% RSLogix 500 project Sesion13_Tarea1_Josue Santana Robledo Corona.RSS, saved by version 8.40.00.08 %
PROJECT "UNTITLED"    % processor: MicroLogix 1200 %

PROGRAM FILES
  LAD 2 "MAIN"  7 rungs
  LAD 3 "ENTRADAS"  7 rungs
  LAD 4 "SALIDAS"  6 rungs
  LAD 5 "MANUAL"  6 rungs
  LAD 6 "AUTOMATICO"  17 rungs
  LAD 7 "HMI"  1 rungs
  LAD 8 "ALARMAS"  1 rungs
  LAD 9 "LS"  4 rungs
  LAD 10 "PARPADEOS"  5 rungs
  LAD 11 "RESET"  3 rungs

DATA FILES
  O0 OUTPUT  4 elements
  I1 INPUT  4 elements
  S2 STATUS  66 elements
  B3 BINARY  4 elements
  T4 TIMER  8 elements
  C5 COUNTER  3 elements
  R6 CONTROL  1 elements
  N7 INTEGER  1 elements
  F8 FLOAT  1 elements

LADDER 2 "MAIN"
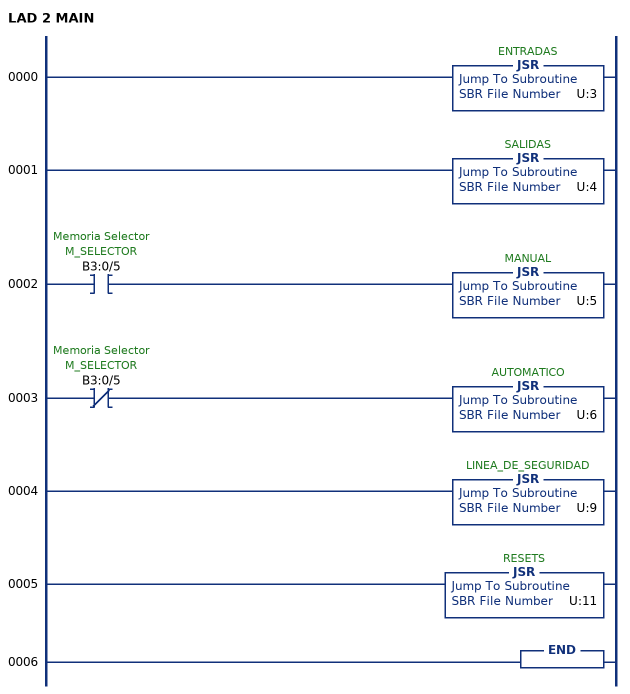
% Rung: 0 %
SOR JSR U:3 EOR
%   U:3  ENTRADAS %
% Rung: 1 %
SOR JSR U:4 EOR
%   U:4  SALIDAS %
% Rung: 2 %
SOR XIC B3:0/5 JSR U:5 EOR
%   B3:0/5  M_SELECTOR  "Memoria Selector" %
%   U:5  MANUAL %
% Rung: 3 %
SOR XIO B3:0/5 JSR U:6 EOR
%   B3:0/5  M_SELECTOR  "Memoria Selector" %
%   U:6  AUTOMATICO %
% Rung: 4 %
SOR JSR U:9 EOR
%   U:9  LINEA_DE_SEGURIDAD %
% Rung: 5 %
SOR JSR U:11 EOR
%   U:11  RESETS %
% Rung: 6 %
SOR END EOR

LADDER 3 "ENTRADAS"
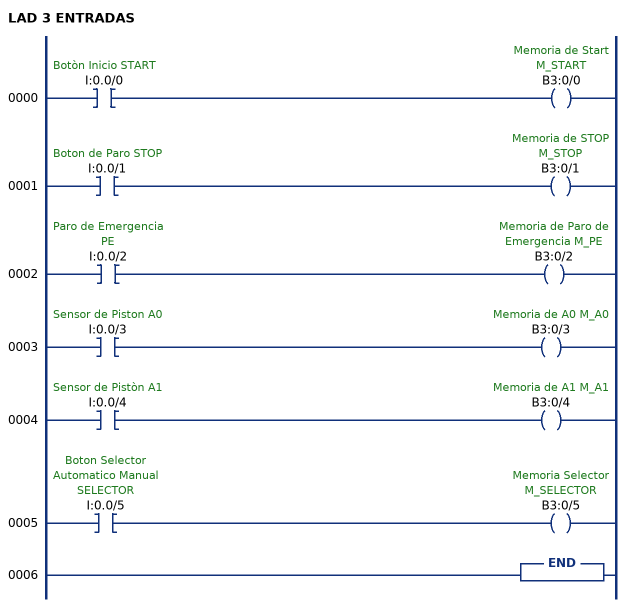
% Rung: 0 %
SOR XIC I:0.0/0 OTE B3:0/0 EOR
%   I:0.0/0  START  "Botòn Inicio" %
%   B3:0/0  M_START  "Memoria de Start" %
% Rung: 1 %
SOR XIC I:0.0/1 OTE B3:0/1 EOR
%   I:0.0/1  STOP  "Boton de Paro" %
%   B3:0/1  M_STOP  "Memoria de STOP" %
% Rung: 2 %
SOR XIC I:0.0/2 OTE B3:0/2 EOR
%   I:0.0/2  PE  "Paro de Emergencia" %
%   B3:0/2  M_PE  "Memoria de Paro de Emergencia" %
% Rung: 3 %
SOR XIC I:0.0/3 OTE B3:0/3 EOR
%   I:0.0/3  A0  "Sensor de Piston" %
%   B3:0/3  M_A0  "Memoria de A0" %
% Rung: 4 %
SOR XIC I:0.0/4 OTE B3:0/4 EOR
%   I:0.0/4  A1  "Sensor de Pistòn" %
%   B3:0/4  M_A1  "Memoria de A1" %
% Rung: 5 %
SOR XIC I:0.0/5 OTE B3:0/5 EOR
%   I:0.0/5  SELECTOR  "Boton Selector Automatico Manual" %
%   B3:0/5  M_SELECTOR  "Memoria Selector" %
% Rung: 6 %
SOR END EOR

LADDER 4 "SALIDAS"
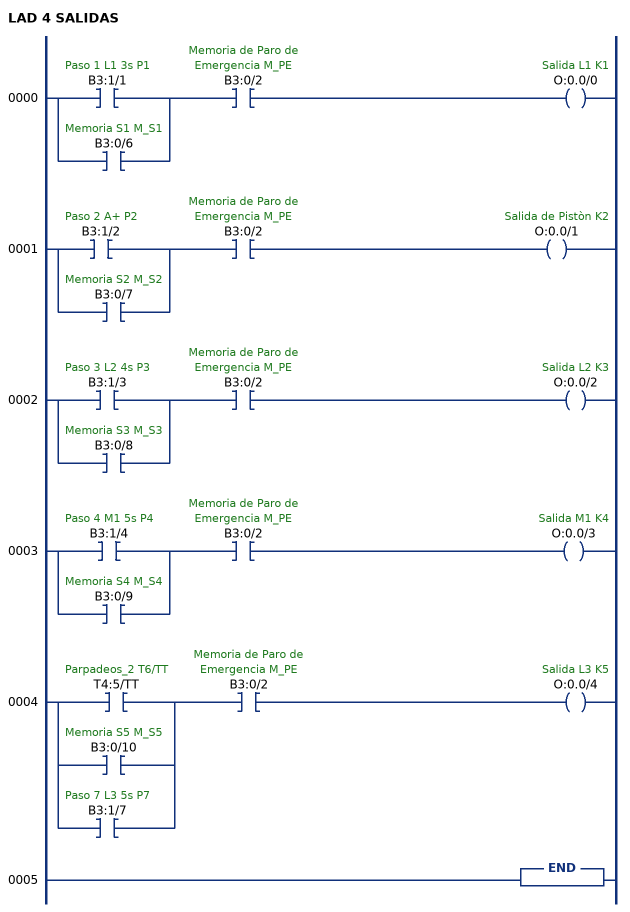
% Rung: 0 %
SOR BST XIC B3:1/1 NXB XIC B3:0/6 BND XIC B3:0/2 OTE O:0.0/0 EOR
%   B3:1/1  P1  "Paso 1 L1 3s" %
%   B3:0/6  M_S1  "Memoria S1" %
%   B3:0/2  M_PE  "Memoria de Paro de Emergencia" %
%   O:0.0/0  K1  "Salida L1" %
% Rung: 1 %
SOR BST XIC B3:1/2 NXB XIC B3:0/7 BND XIC B3:0/2 OTE O:0.0/1 EOR
%   B3:1/2  P2  "Paso 2 A+" %
%   B3:0/7  M_S2  "Memoria S2" %
%   B3:0/2  M_PE  "Memoria de Paro de Emergencia" %
%   O:0.0/1  K2  "Salida de Pistòn" %
% Rung: 2 %
SOR BST XIC B3:1/3 NXB XIC B3:0/8 BND XIC B3:0/2 OTE O:0.0/2 EOR
%   B3:1/3  P3  "Paso 3 L2 4s" %
%   B3:0/8  M_S3  "Memoria S3" %
%   B3:0/2  M_PE  "Memoria de Paro de Emergencia" %
%   O:0.0/2  K3  "Salida L2" %
% Rung: 3 %
SOR BST XIC B3:1/4 NXB XIC B3:0/9 BND XIC B3:0/2 OTE O:0.0/3 EOR
%   B3:1/4  P4  "Paso 4 M1 5s" %
%   B3:0/9  M_S4  "Memoria S4" %
%   B3:0/2  M_PE  "Memoria de Paro de Emergencia" %
%   O:0.0/3  K4  "Salida M1" %
% Rung: 4 %
SOR BST XIC T4:5/TT NXB BST XIC B3:0/10 NXB XIC B3:1/7 BND BND XIC B3:0/2 OTE O:0.0/4 EOR
%   T4:5  T6  "Parpadeos_2" %
%   B3:0/10  M_S5  "Memoria S5" %
%   B3:1/7  P7  "Paso 7 L3 5s" %
%   B3:0/2  M_PE  "Memoria de Paro de Emergencia" %
%   O:0.0/4  K5  "Salida L3" %
% Rung: 5 %
SOR END EOR

LADDER 5 "MANUAL"
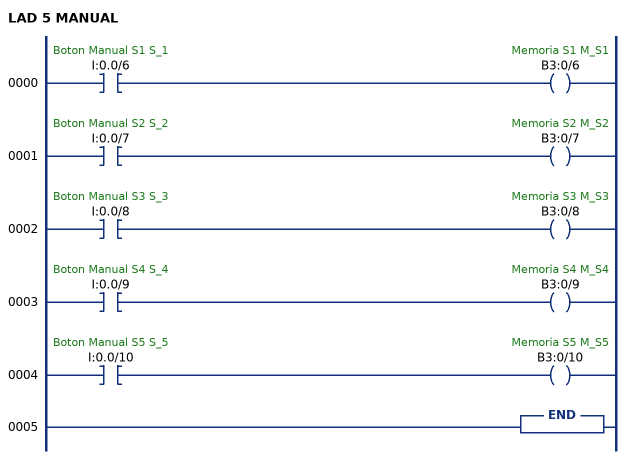
% Rung: 0 %
SOR XIC I:0.0/6 OTE B3:0/6 EOR
%   I:0.0/6  S_1  "Boton Manual S1" %
%   B3:0/6  M_S1  "Memoria S1" %
% Rung: 1 %
SOR XIC I:0.0/7 OTE B3:0/7 EOR
%   I:0.0/7  S_2  "Boton Manual S2" %
%   B3:0/7  M_S2  "Memoria S2" %
% Rung: 2 %
SOR XIC I:0.0/8 OTE B3:0/8 EOR
%   I:0.0/8  S_3  "Boton Manual S3" %
%   B3:0/8  M_S3  "Memoria S3" %
% Rung: 3 %
SOR XIC I:0.0/9 OTE B3:0/9 EOR
%   I:0.0/9  S_4  "Boton Manual S4" %
%   B3:0/9  M_S4  "Memoria S4" %
% Rung: 4 %
SOR XIC I:0.0/10 OTE B3:0/10 EOR
%   I:0.0/10  S_5  "Boton Manual S5" %
%   B3:0/10  M_S5  "Memoria S5" %
% Rung: 5 %
SOR END EOR

LADDER 6 "AUTOMATICO"
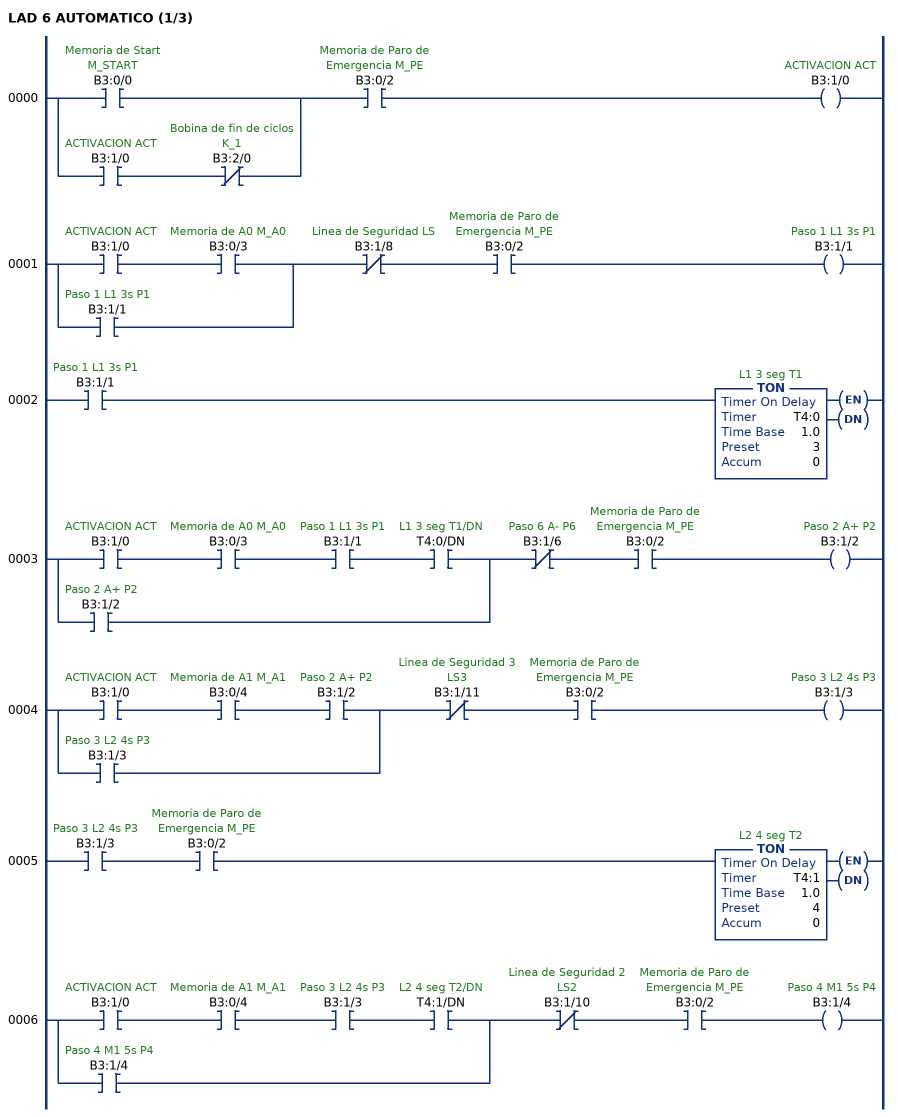
% Rung: 0 %  % edit flag set %
SOR BST XIC B3:0/0 NXB XIC B3:1/0 XIO B3:2/0 BND XIC B3:0/2 OTE B3:1/0 EOR
%   B3:0/0  M_START  "Memoria de Start" %
%   B3:1/0  ACT  "ACTIVACION" %
%   B3:2/0  K_1  "Bobina de fin de ciclos" %
%   B3:0/2  M_PE  "Memoria de Paro de Emergencia" %
% Rung: 1 %
SOR BST XIC B3:1/0 XIC B3:0/3 NXB XIC B3:1/1 BND XIO B3:1/8 XIC B3:0/2 OTE B3:1/1 EOR
%   B3:1/0  ACT  "ACTIVACION" %
%   B3:0/3  M_A0  "Memoria de A0" %
%   B3:1/1  P1  "Paso 1 L1 3s" %
%   B3:1/8  LS  "Linea de Seguridad" %
%   B3:0/2  M_PE  "Memoria de Paro de Emergencia" %
% Rung: 2 %
SOR XIC B3:1/1 TON T4:0 1.0 3 0 EOR
%   B3:1/1  P1  "Paso 1 L1 3s" %
%   T4:0  T1  "L1 3 seg" %
% Rung: 3 %
SOR BST XIC B3:1/0 XIC B3:0/3 XIC B3:1/1 XIC T4:0/DN NXB XIC B3:1/2 BND XIO B3:1/6 XIC B3:0/2 OTE B3:1/2 EOR
%   B3:1/0  ACT  "ACTIVACION" %
%   B3:0/3  M_A0  "Memoria de A0" %
%   B3:1/1  P1  "Paso 1 L1 3s" %
%   T4:0  T1  "L1 3 seg" %
%   B3:1/2  P2  "Paso 2 A+" %
%   B3:1/6  P6  "Paso 6 A-" %
%   B3:0/2  M_PE  "Memoria de Paro de Emergencia" %
% Rung: 4 %
SOR BST XIC B3:1/0 XIC B3:0/4 XIC B3:1/2 NXB XIC B3:1/3 BND XIO B3:1/11 XIC B3:0/2 OTE B3:1/3 EOR
%   B3:1/0  ACT  "ACTIVACION" %
%   B3:0/4  M_A1  "Memoria de A1" %
%   B3:1/2  P2  "Paso 2 A+" %
%   B3:1/3  P3  "Paso 3 L2 4s" %
%   B3:1/11  LS3  "Linea de Seguridad 3" %
%   B3:0/2  M_PE  "Memoria de Paro de Emergencia" %
% Rung: 5 %
SOR XIC B3:1/3 XIC B3:0/2 TON T4:1 1.0 4 0 EOR
%   B3:1/3  P3  "Paso 3 L2 4s" %
%   B3:0/2  M_PE  "Memoria de Paro de Emergencia" %
%   T4:1  T2  "L2 4 seg" %
% Rung: 6 %
SOR BST XIC B3:1/0 XIC B3:0/4 XIC B3:1/3 XIC T4:1/DN NXB XIC B3:1/4 BND XIO B3:1/10 XIC B3:0/2 OTE B3:1/4 EOR
%   B3:1/0  ACT  "ACTIVACION" %
%   B3:0/4  M_A1  "Memoria de A1" %
%   B3:1/3  P3  "Paso 3 L2 4s" %
%   T4:1  T2  "L2 4 seg" %
%   B3:1/4  P4  "Paso 4 M1 5s" %
%   B3:1/10  LS2  "Linea de Seguridad 2" %
%   B3:0/2  M_PE  "Memoria de Paro de Emergencia" %

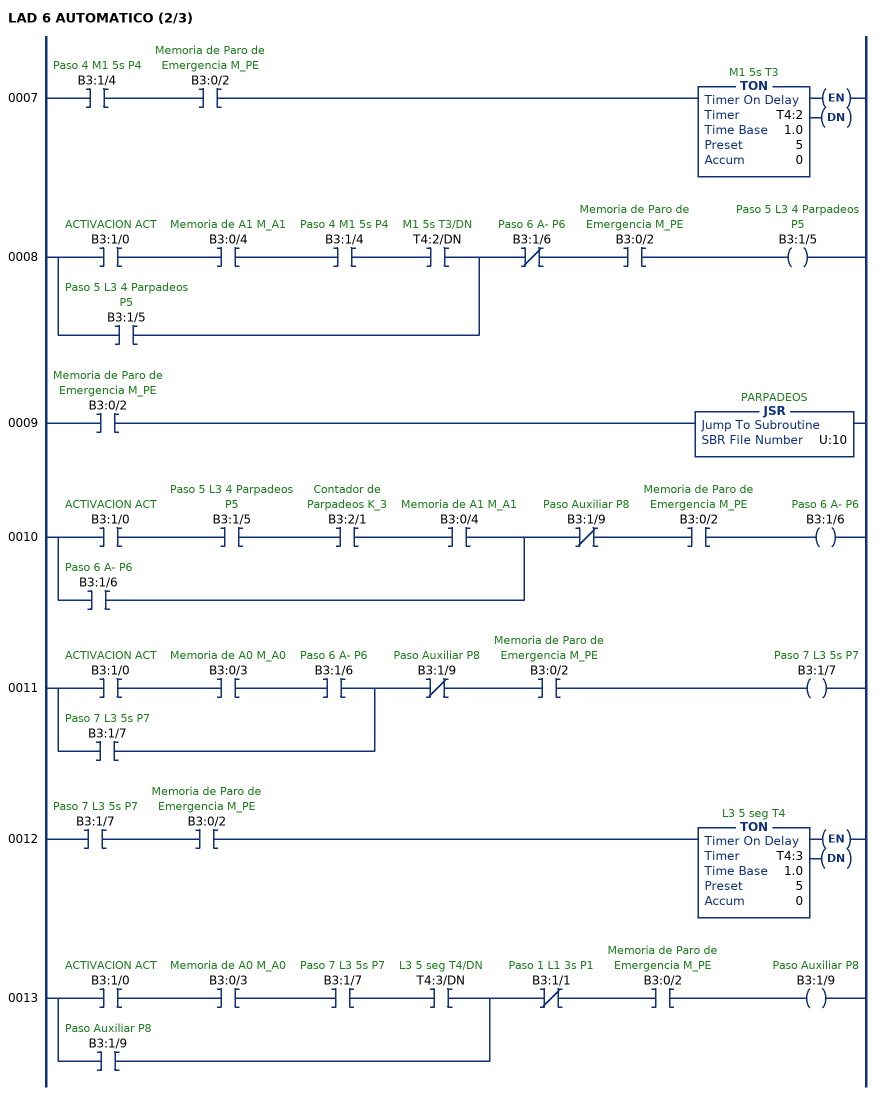
% Rung: 7 %
SOR XIC B3:1/4 XIC B3:0/2 TON T4:2 1.0 5 0 EOR
%   B3:1/4  P4  "Paso 4 M1 5s" %
%   B3:0/2  M_PE  "Memoria de Paro de Emergencia" %
%   T4:2  T3  "M1 5s" %
% Rung: 8 %
SOR BST XIC B3:1/0 XIC B3:0/4 XIC B3:1/4 XIC T4:2/DN NXB XIC B3:1/5 BND XIO B3:1/6 XIC B3:0/2 OTE B3:1/5 EOR
%   B3:1/0  ACT  "ACTIVACION" %
%   B3:0/4  M_A1  "Memoria de A1" %
%   B3:1/4  P4  "Paso 4 M1 5s" %
%   T4:2  T3  "M1 5s" %
%   B3:1/5  P5  "Paso 5 L3 4 Parpadeos" %
%   B3:1/6  P6  "Paso 6 A-" %
%   B3:0/2  M_PE  "Memoria de Paro de Emergencia" %
% Rung: 9 %
SOR XIC B3:0/2 JSR U:10 EOR
%   B3:0/2  M_PE  "Memoria de Paro de Emergencia" %
%   U:10  PARPADEOS %
% Rung: 10 %
SOR BST XIC B3:1/0 XIC B3:1/5 XIC B3:2/1 XIC B3:0/4 NXB XIC B3:1/6 BND XIO B3:1/9 XIC B3:0/2 OTE B3:1/6 EOR
%   B3:1/0  ACT  "ACTIVACION" %
%   B3:1/5  P5  "Paso 5 L3 4 Parpadeos" %
%   B3:2/1  K_3  "Contador de Parpadeos" %
%   B3:0/4  M_A1  "Memoria de A1" %
%   B3:1/6  P6  "Paso 6 A-" %
%   B3:1/9  P8  "Paso Auxiliar" %
%   B3:0/2  M_PE  "Memoria de Paro de Emergencia" %
% Rung: 11 %
SOR BST XIC B3:1/0 XIC B3:0/3 XIC B3:1/6 NXB XIC B3:1/7 BND XIO B3:1/9 XIC B3:0/2 OTE B3:1/7 EOR
%   B3:1/0  ACT  "ACTIVACION" %
%   B3:0/3  M_A0  "Memoria de A0" %
%   B3:1/6  P6  "Paso 6 A-" %
%   B3:1/7  P7  "Paso 7 L3 5s" %
%   B3:1/9  P8  "Paso Auxiliar" %
%   B3:0/2  M_PE  "Memoria de Paro de Emergencia" %
% Rung: 12 %
SOR XIC B3:1/7 XIC B3:0/2 TON T4:3 1.0 5 0 EOR
%   B3:1/7  P7  "Paso 7 L3 5s" %
%   B3:0/2  M_PE  "Memoria de Paro de Emergencia" %
%   T4:3  T4  "L3 5 seg" %
% Rung: 13 %
SOR BST XIC B3:1/0 XIC B3:0/3 XIC B3:1/7 XIC T4:3/DN NXB XIC B3:1/9 BND XIO B3:1/1 XIC B3:0/2 OTE B3:1/9 EOR
%   B3:1/0  ACT  "ACTIVACION" %
%   B3:0/3  M_A0  "Memoria de A0" %
%   B3:1/7  P7  "Paso 7 L3 5s" %
%   T4:3  T4  "L3 5 seg" %
%   B3:1/9  P8  "Paso Auxiliar" %
%   B3:1/1  P1  "Paso 1 L1 3s" %
%   B3:0/2  M_PE  "Memoria de Paro de Emergencia" %

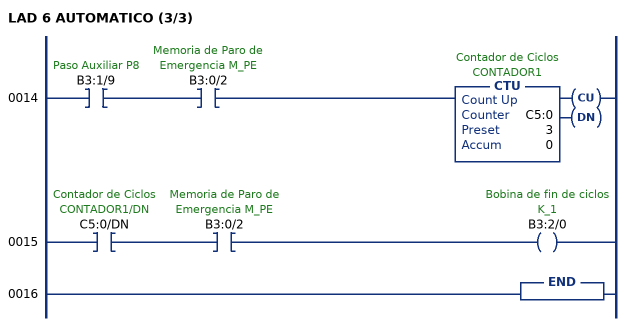
% Rung: 14 %
SOR XIC B3:1/9 XIC B3:0/2 CTU C5:0 3 0 EOR
%   B3:1/9  P8  "Paso Auxiliar" %
%   B3:0/2  M_PE  "Memoria de Paro de Emergencia" %
%   C5:0  CONTADOR1  "Contador de Ciclos" %
% Rung: 15 %
SOR XIC C5:0/DN XIC B3:0/2 OTE B3:2/0 EOR
%   C5:0  CONTADOR1  "Contador de Ciclos" %
%   B3:0/2  M_PE  "Memoria de Paro de Emergencia" %
%   B3:2/0  K_1  "Bobina de fin de ciclos" %
% Rung: 16 %
SOR END EOR

LADDER 9 "LS"
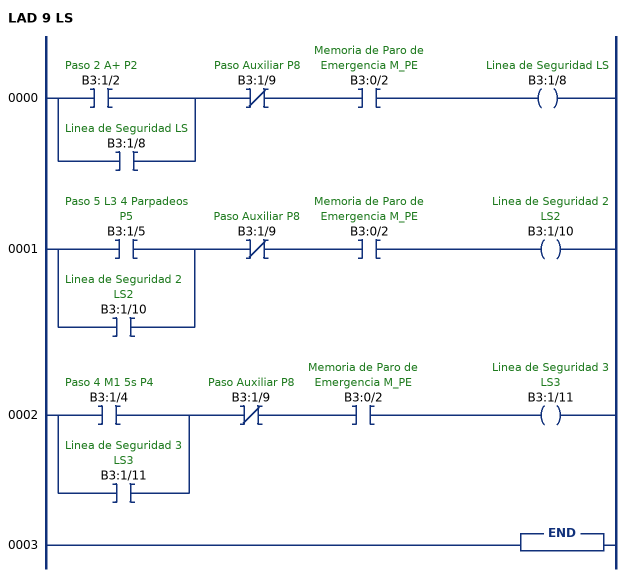
% Rung: 0 %
SOR BST XIC B3:1/2 NXB XIC B3:1/8 BND XIO B3:1/9 XIC B3:0/2 OTE B3:1/8 EOR
%   B3:1/2  P2  "Paso 2 A+" %
%   B3:1/8  LS  "Linea de Seguridad" %
%   B3:1/9  P8  "Paso Auxiliar" %
%   B3:0/2  M_PE  "Memoria de Paro de Emergencia" %
% Rung: 1 %
SOR BST XIC B3:1/5 NXB XIC B3:1/10 BND XIO B3:1/9 XIC B3:0/2 OTE B3:1/10 EOR
%   B3:1/5  P5  "Paso 5 L3 4 Parpadeos" %
%   B3:1/10  LS2  "Linea de Seguridad 2" %
%   B3:1/9  P8  "Paso Auxiliar" %
%   B3:0/2  M_PE  "Memoria de Paro de Emergencia" %
% Rung: 2 %
SOR BST XIC B3:1/4 NXB XIC B3:1/11 BND XIO B3:1/9 XIC B3:0/2 OTE B3:1/11 EOR
%   B3:1/4  P4  "Paso 4 M1 5s" %
%   B3:1/11  LS3  "Linea de Seguridad 3" %
%   B3:1/9  P8  "Paso Auxiliar" %
%   B3:0/2  M_PE  "Memoria de Paro de Emergencia" %
% Rung: 3 %
SOR END EOR

LADDER 10 "PARPADEOS"
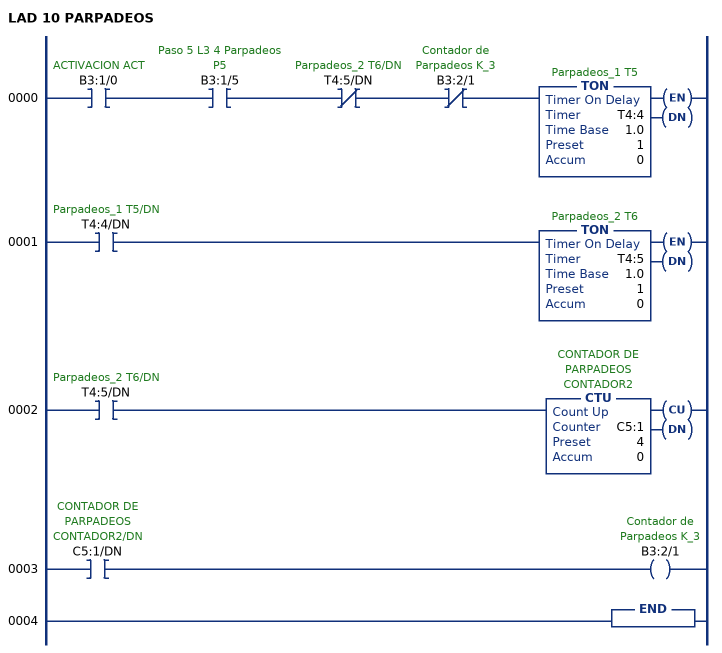
% Rung: 0 %
SOR XIC B3:1/0 XIC B3:1/5 XIO T4:5/DN XIO B3:2/1 TON T4:4 1.0 1 0 EOR
%   B3:1/0  ACT  "ACTIVACION" %
%   B3:1/5  P5  "Paso 5 L3 4 Parpadeos" %
%   T4:5  T6  "Parpadeos_2" %
%   B3:2/1  K_3  "Contador de Parpadeos" %
%   T4:4  T5  "Parpadeos_1" %
% Rung: 1 %
SOR XIC T4:4/DN TON T4:5 1.0 1 0 EOR
%   T4:4  T5  "Parpadeos_1" %
%   T4:5  T6  "Parpadeos_2" %
% Rung: 2 %
SOR XIC T4:5/DN CTU C5:1 4 0 EOR
%   T4:5  T6  "Parpadeos_2" %
%   C5:1  CONTADOR2  "CONTADOR DE PARPADEOS" %
% Rung: 3 %
SOR XIC C5:1/DN OTE B3:2/1 EOR
%   C5:1  CONTADOR2  "CONTADOR DE PARPADEOS" %
%   B3:2/1  K_3  "Contador de Parpadeos" %
% Rung: 4 %
SOR END EOR

LADDER 11 "RESET"
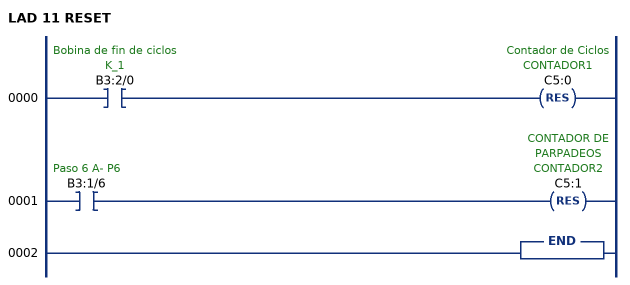
% Rung: 0 %
SOR XIC B3:2/0 RES C5:0 EOR
%   B3:2/0  K_1  "Bobina de fin de ciclos" %
%   C5:0  CONTADOR1  "Contador de Ciclos" %
% Rung: 1 %
SOR XIC B3:1/6 RES C5:1 EOR
%   B3:1/6  P6  "Paso 6 A-" %
%   C5:1  CONTADOR2  "CONTADOR DE PARPADEOS" %
% Rung: 2 %
SOR END EOR

OTHER DOCUMENTED ADDRESSES
  B3:2/2  K_2  "Parpadeos"
  C5:2  CONTADOR3  "Contador de Parpadeos1"
  T4:6  T7  "Primeros Parpadeos_1"
  T4:7  T8  "Primeros Parpadeos_2"

DATA TABLE (non-zero values as saved)
DATA B3
% B3:0 % 0X0016 0X0D25 0X0000 0X0000
DATA T4
% .PRE .ACC %
% T4:0 % 3 0
% T4:1 % 4 0
% T4:2 % 5 0
% T4:3 % 5 0
% T4:4 % 1 0
% T4:5 % 1 0
% T4:6 % 1 0
% T4:7 % 1 0
DATA C5
% .PRE .ACC %
% C5:0 % 3 0
% C5:1 % 4 0
% C5:2 % 4 0
